TYPE ST_Dynamics :
STRUCT
  Velocity : LREAL;
  Accleration : LREAL;
  Deceleration : LREAL;
END_STRUCT
END_TYPE

(* stored: Version 1.1.0.1
   DUT ST_Dynamics: Id {304e4601-fb73-42f1-8555-efd083442923} *)
